   VAR
      s_FB_TRCV {InstructionName := 'TRCV'; LibVersion := '4.0'; ExternalAccessible := 'False'; ExternalVisible := 'False'; ExternalWritable := 'False'; S7_SetPoint := 'False'} : TRCV;   // Siemens "TRCV" block - to receive the data from TCPIP socket
      ss_TRCV { ExternalAccessible := 'False'; ExternalVisible := 'False'; ExternalWritable := 'False'} : Struct   // TRCV block interface structure
         Enable { ExternalAccessible := 'False'; ExternalVisible := 'False'; ExternalWritable := 'False'} : Bool;   //      TRCV - Enable
         NDR { ExternalAccessible := 'False'; ExternalVisible := 'False'; ExternalWritable := 'False'} : Bool;   //      TRCV - New data available
         Busy { ExternalAccessible := 'False'; ExternalVisible := 'False'; ExternalWritable := 'False'} : Bool;   //      TRCV - Busy
         Error { ExternalAccessible := 'False'; ExternalVisible := 'False'; ExternalWritable := 'False'} : Bool;   //      TRCV - Error
         Status { ExternalAccessible := 'False'; ExternalVisible := 'False'; ExternalWritable := 'False'} : Word;   //      TRCV - Status
         ReceivedLength { ExternalAccessible := 'False'; ExternalVisible := 'False'; ExternalWritable := 'False'} : UDInt;   //      TRCV - Received length
         Data { ExternalAccessible := 'False'; ExternalVisible := 'False'; ExternalWritable := 'False'} : Array[0..999] of Char;   //      TRCV - Data
      END_STRUCT;
      s_UDT_MessageArray { ExternalAccessible := 'False'; ExternalVisible := 'False'; ExternalWritable := 'False'; S7_SetPoint := 'False'} : "UDT_Message";   // Message byte array
      s_UDT_MessagePartArray { ExternalAccessible := 'False'; ExternalVisible := 'False'; ExternalWritable := 'False'; S7_SetPoint := 'False'} : "UDT_Message";   // Part of the message byte array
      ss_Status { ExternalAccessible := 'False'; ExternalVisible := 'False'; ExternalWritable := 'False'} : Struct   // Status structure
         ErrorCode { ExternalAccessible := 'False'; ExternalVisible := 'False'; ExternalWritable := 'False'} : Struct   // Error code structure
            TRCV { ExternalAccessible := 'False'; ExternalVisible := 'False'; ExternalWritable := 'False'} : Word;   //     Siemens TRCV error code - Check documentation
         END_STRUCT;
         FIFOReceiveStatus { ExternalAccessible := 'False'; ExternalVisible := 'False'; ExternalWritable := 'False'} : "UDT_FifoStatus";   // Receive FIFO status structure
         FIFOReceiveError { ExternalAccessible := 'False'; ExternalVisible := 'False'; ExternalWritable := 'False'; S7_SetPoint := 'True'} : Bool;   // Receive FIFO error
         FIFOReceiveWarning { ExternalAccessible := 'False'; ExternalVisible := 'False'; ExternalWritable := 'False'; S7_SetPoint := 'True'} : Bool;   // Receive  FIFO warning
         ReceiveError { ExternalAccessible := 'False'; ExternalVisible := 'False'; ExternalWritable := 'False'} : Bool;   // TRCV block operation error - Check TRCVStatus
      END_STRUCT;
      sui_ReceivedMessagesOffset { ExternalAccessible := 'False'; ExternalVisible := 'False'; ExternalWritable := 'False'} : Int;   // Received message offset
      sui_ReceivedMessageLength { ExternalAccessible := 'False'; ExternalVisible := 'False'; ExternalWritable := 'False'} : UInt;   // Received message length
      sui_NumberOfReceivedMessages { ExternalAccessible := 'False'; ExternalVisible := 'False'; ExternalWritable := 'False'} : UInt;   // Number of received messages in one frame
      sui_ReceivedMessagePartLength { ExternalAccessible := 'False'; ExternalVisible := 'False'; ExternalWritable := 'False'} : UInt;   // Length of the part of received message
      si_MaximumMessageLength { ExternalAccessible := 'False'; ExternalVisible := 'False'; ExternalWritable := 'False'} : Int;   // Maximum message length
      sx_ReceivedMessagePart { ExternalAccessible := 'False'; ExternalVisible := 'False'; ExternalWritable := 'False'} : Bool;   // Received part of the message
      sx_STXFound { ExternalAccessible := 'False'; ExternalVisible := 'False'; ExternalWritable := 'False'} : Bool;   // STX in message is found
   END_VAR

   VAR_TEMP
      ti_LC_MessageChars : Int;   //  Message chars loop counter
   END_VAR

   VAR CONSTANT
      cc_STX : Char := '$02';   // Start of the message sign
      cc_EXT : Char := '$03';   // End of the message sign
      cc_NULL : Char := '$00';   // Null sign
   END_VAR


BEGIN
	(*
	----------------------------------------------------------------------------------------

	Version history:
	Date        | Version   | Author        | Remark
	----------------------------------------------------------------------------------------
	25/10/2021  | 1.0       | J. Krawczuk   | Initial version TIA 16
	17/11/2021  | 1.2       | M. Piela      | Interface changes
	21/02/2023  | 4.0       | F.Baten       | 4.0 Release TIA 17.5
	13/03/2024  | 4.1       | S. Nieświec   | 4.1 Release TIA 18
	02/05/2024  | 4.2       | J.Majer      | Datatype conversions changed from automatic to explicit, to accomodate IEC 61131-3 standard
	*)

	REGION 1 – Update FIFO header status bits

	    // Mode 'S' - FIFO register status update.
	    "FC_Fifo"(ic_Mode := 'S',
	              qUDT_Status => #ss_Status.FIFOReceiveStatus,
	              qx_Error => #ss_Status.FIFOReceiveError,
	              qx_Warning => #ss_Status.FIFOReceiveWarning,
	              iqv_Data := #s_UDT_MessageArray,
	              iqUDT_FifoHeader := #iqUDT_FifoHeader,
	              iqv_DataBuffer := #iqv_FifoData);

	END_REGION

	REGION 2 – Maximum number of message arrays elements

	    #si_MaximumMessageLength := "FC_GetNrOfArrayEl"(iv_Array := #s_UDT_MessageArray.Character);

	END_REGION

	REGION 3 – Receive enable

	    // Allow receiving if the connection is established and there are no FIFO errors.
	    #ss_TRCV.Enable :=
	    #ix_EnableReceive
	    AND NOT #ss_Status.FIFOReceiveError;

	END_REGION

	REGION 4 – Receive data

	    // Data received in an ADHOC mode - data available immediately.
	    #s_FB_TRCV(EN_R := #ss_TRCV.Enable,
	               ID := #iUDT_Connection.ID,
	               LEN := 0,
	               ADHOC := TRUE,
	               NDR => #ss_TRCV.NDR,
	               BUSY => #ss_TRCV.Busy,
	               ERROR => #ss_TRCV.Error,
	               STATUS => #ss_TRCV.Status,
	               RCVD_LEN => #ss_TRCV.ReceivedLength,
	               DATA := #ss_TRCV.Data);

	END_REGION

	REGION 5 – Received data handling

	    // Receiving data was successful.
	    IF #ss_TRCV.NDR
	        AND NOT #ss_TRCV.Busy
	        AND NOT #ss_TRCV.Error
	        AND #ss_TRCV.ReceivedLength > 0

	    THEN

	        REGION 5.1 – Initialization

	            #sui_ReceivedMessageLength := 0;
	            #sui_ReceivedMessagesOffset := 0;
	            #sui_NumberOfReceivedMessages := 0;

	        END_REGION

	        REGION 5.2 – Received part of the message

	            // Move part of the messages into a buffer if available.
	            IF #sx_ReceivedMessagePart
	            THEN
	                #s_UDT_MessageArray := #s_UDT_MessagePartArray;
	            END_IF;

	        END_REGION

	        REGION 5.3 – Message handling

	            FOR #ti_LC_MessageChars := 0 TO (UDINT_TO_INT(#ss_TRCV.ReceivedLength) - 1) DO
	                // Message length validation.
	                IF #sui_ReceivedMessageLength <= #si_MaximumMessageLength
	                THEN
	                    // First termination sign found.
	                    IF (#ss_TRCV.Data[#ti_LC_MessageChars] = #cc_STX)
	                        AND NOT #sx_STXFound
	                    THEN
	                        #sx_STXFound := TRUE;
	                        #sui_ReceivedMessagesOffset := #ti_LC_MessageChars;

	                    ELSIF (#ss_TRCV.Data[#ti_LC_MessageChars] = #cc_STX)
	                        AND #sx_STXFound
	                    THEN
	                        // Increment invalid meassage statistic.
	                        #iqUDT_Statistics.InvalidMsg += 1;
	                        #sx_STXFound := FALSE;
	                    END_IF;

	                    // STX is found.
	                    IF #sx_STXFound
	                    THEN
	                        // Increment received message length.
	                        #sui_ReceivedMessageLength += 1;

	                        // End of the message sign is found.
	                        IF #ss_TRCV.Data[#ti_LC_MessageChars] = #cc_EXT
	                        THEN
	                            // Move received message to the message array.
	                            MOVE_BLK(IN := #ss_TRCV.Data[#sui_ReceivedMessagesOffset],
	                                     COUNT := #sui_ReceivedMessageLength,
	                                     OUT => #s_UDT_MessageArray.Character[#sui_ReceivedMessagePartLength]);

	                            // Clear not used message array characters.
	                            IF (#sui_ReceivedMessageLength + #sui_ReceivedMessagePartLength) < #si_MaximumMessageLength
	                            THEN
	                                FILL_BLK(IN := #cc_NULL,
	                                         COUNT := INT_TO_ULINT(#si_MaximumMessageLength) -
	                                         UDINT_TO_ULINT(#sui_ReceivedMessageLength) + #sui_ReceivedMessagePartLength,
	                                         OUT => #s_UDT_MessageArray.Character[#sui_ReceivedMessageLength + #sui_ReceivedMessagePartLength]);
	                            END_IF;

	                            // Mode 'W' - Write FIFO record.
	                            "FC_Fifo"(ic_Mode := 'W',
	                                      qUDT_Status => #ss_Status.FIFOReceiveStatus,
	                                      qx_Error => #ss_Status.FIFOReceiveError,
	                                      qx_Warning => #ss_Status.FIFOReceiveWarning,
	                                      iqv_Data := #s_UDT_MessageArray,
	                                      iqUDT_FifoHeader := #iqUDT_FifoHeader,
	                                      iqv_DataBuffer := #iqv_FifoData);

	                            // Increment received message count.
	                            #sui_NumberOfReceivedMessages += 1;
	                            // Initialize variables.
	                            #sui_ReceivedMessageLength := 0;
	                            #sui_ReceivedMessagePartLength := 0;
	                            #sx_ReceivedMessagePart := FALSE;
	                            #sx_STXFound := FALSE;

	                        END_IF;
	                    END_IF;
	                END_IF;
	            END_FOR;

	        END_REGION

	        REGION 5.4 – Part of the message preparation

	            // Only the part of the message is received.
	            IF (#ss_TRCV.Data[UDINT_TO_INT(#ss_TRCV.ReceivedLength) - 1] <> #cc_EXT            // Last received sign is not a termination sing
	                AND #sui_ReceivedMessageLength < #si_MaximumMessageLength)       // Message length valid
	                AND #sx_STXFound
	            THEN
	                // Clear not used message array characters.
	                FILL_BLK(IN := #cc_NULL,
	                         COUNT := INT_TO_ULINT(#si_MaximumMessageLength) -
	                         UDINT_TO_ULINT(#sui_ReceivedMessageLength),
	                         OUT => #s_UDT_MessagePartArray.Character[#sui_ReceivedMessageLength]);

	                // Move part of the message into a buffer.
	                MOVE_BLK(IN := #ss_TRCV.Data[#sui_ReceivedMessagesOffset],
	                         COUNT := #sui_ReceivedMessageLength,
	                         OUT => #s_UDT_MessagePartArray.Character[0]);

	                // Set the part of the message received bit and move length of the received message into the length of the part of the message variable.
	                #sx_ReceivedMessagePart := TRUE;
	                #sui_ReceivedMessagePartLength := #sui_ReceivedMessageLength;
	            END_IF;

	        END_REGION

	    END_IF;

	END_REGION

	REGION 6 – Status

	    REGION 6.1 - Block status

	        // Receive error.
	        #ss_Status.ReceiveError := #ss_TRCV.Error;

	        // Parametrization collective error output.
	        #qx_Error :=
	        #ss_Status.FIFOReceiveError
	        OR #ss_Status.ReceiveError;

	        // Parametrization collective warning output.
	        #qx_Warning := #ss_Status.FIFOReceiveWarning;

	    END_REGION

	    REGION 6.2 - Error code preparation

	        IF (#ss_TRCV.#Status > 16#8000)
	            OR (#ss_TRCV.#Status = 16#0)
	        THEN
	            #ss_Status.ErrorCode.TRCV := #ss_TRCV.#Status;
	        END_IF;

	    END_REGION
	END_REGION
END_FUNCTION_BLOCK

FUNCTION_BLOCK "FB_FedExHeartbeat"
TITLE = FB_Heartbeat
{ S7_Optimized_Access := 'TRUE' }
AUTHOR : MHSE
FAMILY : UPS_SpecificCommunication
VERSION : 3.0
// ATTRIBUTES
// AUTO_NUMBER = True
// BLOCK_NUMBER = 74
// END_ATTRIBUTES
//Function block to send and monitor the UPS heartbeat message.
   VAR_INPUT
      iudi_HeartbeatTimeout { ExternalAccessible := 'False'; ExternalVisible := 'False'; ExternalWritable := 'False'} : UDInt;   // Time after which block show heartbeat error
      iudi_HeartbeatInterval { ExternalAccessible := 'False'; ExternalVisible := 'False'; ExternalWritable := 'False'} : UDInt;   // Heartbeat send interval
      ix_Server { ExternalAccessible := 'False'; ExternalVisible := 'False'; ExternalWritable := 'False'} : Bool;   // PLC is Server ( True = Server )
      ix_EnableSend { ExternalAccessible := 'False'; ExternalVisible := 'False'; ExternalWritable := 'False'} : Bool;   // Enable heartbeat message send
      ix_ResetData { ExternalAccessible := 'False'; ExternalVisible := 'False'; ExternalWritable := 'False'} : Bool;   // Reset statistics
   END_VAR

   VAR_OUTPUT
      qx_HeartbeatOK { ExternalAccessible := 'False'; ExternalVisible := 'False'; ExternalWritable := 'False'} : Bool;   // Heartbeat ok
      qx_Error { ExternalAccessible := 'False'; ExternalVisible := 'False'; ExternalWritable := 'False'} : Bool;   // Collective error output
      qx_Warning { ExternalAccessible := 'False'; ExternalVisible := 'False'; ExternalWritable := 'False'} : Bool;   // Collective warning output
   END_VAR

   VAR_IN_OUT
      iqUDT_FifoHeader : "UDT_FifoHeader";   // FIFO header
      iqa_FifoData : Array[*] of "UDT_Message";   // FIFO data
      iqUDT_Statistics : "UDT_FedExHeartbeatStatistics";   // Heartbeat Statistics
      iqx_Heartbeat { ExternalAccessible := 'False'; ExternalVisible := 'False'; ExternalWritable := 'False'} : Bool;   // Heartbreat received
      iqx_ResetWritingTimer { ExternalAccessible := 'False'; ExternalVisible := 'False'; ExternalWritable := 'False'} : Bool;   // Any message received, do not send Heartbeat
      iqx_ResetListeningTimer { ExternalAccessible := 'False'; ExternalVisible := 'False'; ExternalWritable := 'False'} : Bool;   // Any message received, reset timeout timer
      iqx_SendLS { ExternalAccessible := 'False'; ExternalVisible := 'False'; ExternalWritable := 'False'} : Bool;   // Close the connection
      iqx_Reconnect { ExternalAccessible := 'False'; ExternalVisible := 'False'; ExternalWritable := 'False'} : Bool;   // Reconnect command
   END_VAR

   VAR
      sR_TRIG_EnableSend {InstructionName := 'R_TRIG'; LibVersion := '1.0'; ExternalAccessible := 'False'; ExternalVisible := 'False'; ExternalWritable := 'False'; S7_SetPoint := 'False'} : R_TRIG;   // Siemens "R_TRIG" - to prepare the rising edge trigger on "ix_EnableSend" signal
      sUDT_MessageArray { ExternalAccessible := 'False'; ExternalVisible := 'False'; ExternalWritable := 'False'; S7_SetPoint := 'False'} : "UDT_Message";   // Message character array
      sa_Status { ExternalAccessible := 'False'; ExternalVisible := 'False'; ExternalWritable := 'False'} : Struct   // Status structure
         FIFOStatus { ExternalAccessible := 'False'; ExternalVisible := 'False'; ExternalWritable := 'False'} : "UDT_FifoStatus";
         FIFOError { ExternalAccessible := 'False'; ExternalVisible := 'False'; ExternalWritable := 'False'; S7_SetPoint := 'True'} : Bool;   // FIFO data buffer full
         FIFOWarning { ExternalAccessible := 'False'; ExternalVisible := 'False'; ExternalWritable := 'False'; S7_SetPoint := 'True'} : Bool;   // FIFO error
         HeartbeatOk { ExternalAccessible := 'False'; ExternalVisible := 'False'; ExternalWritable := 'False'} : Bool;   // FIFO warning
         InvalidTimeInterval { ExternalAccessible := 'False'; ExternalVisible := 'False'; ExternalWritable := 'False'} : Bool;   // Heartbeat ok
         InvalidTimeout { ExternalAccessible := 'False'; ExternalVisible := 'False'; ExternalWritable := 'False'} : Bool;   // Heartbeat time interval lower than zero
         InvalidMsgArraySize { ExternalAccessible := 'False'; ExternalVisible := 'False'; ExternalWritable := 'False'} : Bool;   // Heartbeat timeout lower than zero or lower than heartbeat time interval
      END_STRUCT;
      sFB_HeartbeatPulse { ExternalAccessible := 'False'; ExternalVisible := 'False'; ExternalWritable := 'False'; S7_SetPoint := 'False'} : "FB_TimerOnOffDelay";   // Sending Heartbeat timer
      sFB_Timer_HeartbeatCheck { ExternalAccessible := 'False'; ExternalVisible := 'False'; ExternalWritable := 'False'; S7_SetPoint := 'False'} : "FB_TimerOnOffDelay";   // MHS "FB_TimerOnOffDelay" - to measure the time of  missing Hearbeat
      ss_Message { ExternalAccessible := 'False'; ExternalVisible := 'False'; ExternalWritable := 'False'} : String;   // Message character string
      sui_MsgArrayElNr { ExternalAccessible := 'False'; ExternalVisible := 'False'; ExternalWritable := 'False'} : UInt;   // Invalid message array size
      si_MaxMsgLen { ExternalAccessible := 'False'; ExternalVisible := 'False'; ExternalWritable := 'False'} : Int;   // Maximum message length
      si_MsgLen { ExternalAccessible := 'False'; ExternalVisible := 'False'; ExternalWritable := 'False'} : Int;   // String character message length
      si_LostMsg { ExternalAccessible := 'False'; ExternalVisible := 'False'; ExternalWritable := 'False'} : Int;   // Number of lost heartbeat messages
      sx_HeartbeatPulse { ExternalAccessible := 'False'; ExternalVisible := 'False'; ExternalWritable := 'False'} : Bool;   // Heartbeat pulse
      sx_HeartbeatOk { ExternalAccessible := 'False'; ExternalVisible := 'False'; ExternalWritable := 'False'} : Bool;   // Heartbeat ok
      sx_MsgLost { ExternalAccessible := 'False'; ExternalVisible := 'False'; ExternalWritable := 'False'} : Bool;   // Message lost
      sx_HeartbeatCheck { ExternalAccessible := 'False'; ExternalVisible := 'False'; ExternalWritable := 'False'} : Bool;   // Heartbeat check
   END_VAR

   VAR CONSTANT
      cc_STX : Char := '$02';   // Start of the text
      cc_ETX : Char := '$03';   // End of the text
      cc_NULL : Char := '$00';   // NULL sign
      cs_Length : String := '0006';   // Legth of the message
      cs_MessageType : String := 'HB';   // Message type
   END_VAR


BEGIN
	(*
	----------------------------------------------------------------------------------------

	Version history:
	Date        | Version   | Author        | Remark
	----------------------------------------------------------------------------------------
	29/06/2021  | 0.1       | F.Baten       | First release 16.0
	05/04/2022  | 0.2       | K.Pokorski    | Review
	21/02/2023  | 4.0       | F.Baten       | 4.0 Release TIA 17.5
	*)

	REGION 1 – FIFO header status update

	    // Mode 'S' - FIFO register status update
	    "FC_Fifo"(ic_Mode := 'S',
	              qUDT_Status => #sa_Status.FIFOStatus,
	              qx_Error => #sa_Status.FIFOError,
	              qx_Warning => #sa_Status.FIFOWarning,
	              iqv_Data := #sUDT_MessageArray,
	              iqUDT_FifoHeader := #iqUDT_FifoHeader,
	              iqv_DataBuffer := #iqa_FifoData);


	END_REGION

	REGION 2 – Heartbeat time interval and timeout validation
	    IF NOT #ix_Server
	    THEN
	        #sa_Status.InvalidTimeInterval := #iudi_HeartbeatInterval <= 0;

	        #sa_Status.InvalidTimeout := #iudi_HeartbeatTimeout <= 0
	        OR #iudi_HeartbeatTimeout <= #iudi_HeartbeatInterval;
	    END_IF;

	END_REGION

	REGION 3 – Heartbeat pulse generation

	    IF (NOT #sa_Status.InvalidTimeInterval                  // Preset heartbeat time interval is valid
	        AND NOT #sa_Status.InvalidTimeout)                  // Timeout is valid
	        AND NOT #ix_Server
	    THEN

	        #sFB_HeartbeatPulse(iudi_OnDelayTime := #iudi_HeartbeatInterval,
	                            iudi_OffDelayTime := 0,
	                            ix_SignalToDelay := NOT #iqx_ResetWritingTimer,
	                            qx_DelayedSignal => #sx_HeartbeatPulse);

	        IF #sx_HeartbeatPulse THEN
	            #iqx_ResetWritingTimer := TRUE;
	        ELSE
	            #iqx_ResetWritingTimer := FALSE;
	        END_IF;

	    END_IF;

	    // Reset heartbeat send request if PLC is a server
	    IF #ix_Server
	    THEN
	        #sx_HeartbeatPulse := #iqx_Heartbeat;
	        //  #iqx_Heartbeat := FALSE;
	    END_IF;
	END_REGION

	REGION 4 – Heartbeat message preparation

	    IF (NOT #iqUDT_FifoHeader.Status.Full)                 // FIFO isn't full
	    THEN

	        IF (#sx_HeartbeatPulse                              // Heartbeat pulse available
	            AND #ix_EnableSend                              // Send is enable
	            AND NOT #sa_Status.FIFOError)                   // No FIFO error
	        THEN
	            REGION 4.1 – Message preparation

	                // Heartbeat message composing according to the structure: STX,00,06,HB,ETX
	                #ss_Message := CONCAT(IN1 := #cc_STX,               // Start of message
	                                      IN2 := #cs_Length,            // message length
	                                      IN3 := #cs_MessageType,       // Heartbeat
	                                      IN4 := #cc_ETX);              // End of message

	            END_REGION

	            REGION 4.2 – Maximum number of the message characters

	                #si_MaxMsgLen := "FC_GetNrOfArrayEl"(iv_Array := #sUDT_MessageArray.Character);

	            END_REGION

	            REGION 4.3 – Length of the complete message

	                #si_MsgLen := LEN(#ss_Message);

	            END_REGION

	            REGION 4.4 –  Message array size validation

	                #sa_Status.InvalidMsgArraySize := #si_MsgLen > #si_MaxMsgLen;

	            END_REGION

	            REGION 4.5 –  Message character string conversion to a message array of characters

	                IF (NOT #sa_Status.InvalidMsgArraySize)     // Message character array size is valid
	                THEN

	                    Strg_TO_Chars(Strg := #ss_Message,
	                                  pChars := 0,
	                                  Cnt => #sui_MsgArrayElNr,
	                                  Chars := #sUDT_MessageArray.Character);

	                END_IF;

	            END_REGION

	            REGION 4.6 – Clearing remaining characters in the message character array

	                IF (NOT #sa_Status.InvalidMsgArraySize)     // Message character array size is valid
	                THEN

	                    // Filling up not used message character array elements with '$00' (ASCII - 16#00)
	                    FILL_BLK(IN := #cc_NULL,
	                             COUNT := UINT_TO_ULINT(INT_TO_UINT(#si_MaxMsgLen) - #sui_MsgArrayElNr),
	                             OUT => #sUDT_MessageArray.Character[#sui_MsgArrayElNr]);

	                END_IF;

	            END_REGION

	            REGION 4.7 – Message write into a FIFO register

	                IF (#ix_EnableSend                          // Heartbeat send enable
	                    AND NOT #sa_Status.InvalidMsgArraySize) // Message character array size is valid
	                THEN

	                    // Mode 'W' - Write FIFO record
	                    "FC_Fifo"(ic_Mode := 'W',
	                              qUDT_Status => #sa_Status.FIFOStatus,
	                              qx_Error => #sa_Status.FIFOError,
	                              qx_Warning => #sa_Status.FIFOWarning,
	                              iqv_Data := #sUDT_MessageArray,
	                              iqUDT_FifoHeader := #iqUDT_FifoHeader,
	                              iqv_DataBuffer := #iqa_FifoData);
	                END_IF;

	            END_REGION

	        END_IF;

	        // In case of FIFO full, the FIFO full error bit and FIFO collective error bit are set
	    ELSE

	        #sa_Status.FIFOError := TRUE;
	        #sa_Status.FIFOStatus.FifoFull := TRUE;

	    END_IF;

	END_REGION

	REGION 5 – Heartbeat monitoring
	    // IF NOT #ix_Server
	    // THEN
	    IF (NOT #sa_Status.InvalidTimeInterval                  // Time interval is valid
	        AND NOT #sa_Status.InvalidTimeout                   // Timeout is  valid
	        AND NOT #sa_Status.InvalidMsgArraySize)             // Message character array size is valid

	    THEN

	        #sR_TRIG_EnableSend(CLK := #ix_EnableSend);

	        // Reset heartbeat ok
	        IF (NOT #ix_EnableSend)                             // Heartbeat send not enable
	        THEN
	            #iqx_SendLS := FALSE;
	            #sx_HeartbeatOk := FALSE;

	        END_IF;

	        // Clear auxiliary variables
	        IF (#iqx_Heartbeat                                  // Hearbeat message received
	            AND #ix_EnableSend)                             // Heartbeat send enable
	        THEN

	            #si_LostMsg := 0;                               // Lost messages counter
	            #sx_MsgLost := FALSE;                           // Message lost bit
	            #sx_HeartbeatOk := TRUE;                        // HeartbeatOk bit

	        END_IF;

	        // Time measurement of a missing heartbeat
	        #sFB_Timer_HeartbeatCheck(ix_SignalToDelay := #iqx_Heartbeat           // Heartbeat signal
	                                  OR #sx_MsgLost                               // Message lost
	                                  OR #sR_TRIG_EnableSend.Q                    // Enable send trigger
	                                  OR #iqx_ResetListeningTimer,                 // Any message received in this socket
	                                  iudi_OnDelayTime := 0,
	                                  iudi_OffDelayTime := #iudi_HeartbeatTimeout,
	                                  qx_DelayedSignal => #sx_HeartbeatCheck);

	        #iqx_Heartbeat := FALSE;
	        #sx_MsgLost := FALSE;
	        #iqx_ResetListeningTimer := FALSE;

	        // Increment lost messages counter and set lost message bit
	        IF (NOT #sx_HeartbeatCheck                          // Heartbeat not checked
	            AND NOT #iqx_Reconnect                          // No reconnect command
	            AND #ix_EnableSend)                             // Send is enable
	        THEN

	            // Send LS, re-establish connection, increment statistics and signalize heartbeat error

	            #iqx_SendLS := TRUE;
	            #iqUDT_Statistics.ConLost += 1;
	            #si_LostMsg := 0;
	            #sx_MsgLost := FALSE;
	            #sx_HeartbeatOk := FALSE;

	        END_IF;

	        // Configuration error occured
	    ELSE

	        #sx_HeartbeatOk := FALSE;

	    END_IF;
	    // END_IF;

	END_REGION

	REGION 6 – Statistics

	    IF #iqUDT_FifoHeader.Status.Full
	        AND #sx_HeartbeatPulse
	    THEN
	        #iqUDT_Statistics.MsgNotSent += 1;

	    END_IF;

	    IF (#ix_ResetData)                                      // Reset statistics request
	    THEN
	        #iqUDT_Statistics.ConLost := 0;
	        #iqUDT_Statistics.MsgNotSent := 0;

	    END_IF;

	END_REGION

	REGION 7 – Status

	    // Hearbeat ok output
	    #qx_HeartbeatOK := #sx_HeartbeatOk;

	    // Parametrization collective error output
	    #qx_Error :=
	    #sa_Status.InvalidTimeInterval                          // Invalid time interval
	    OR #sa_Status.InvalidTimeout                            // Invalid timeout
	    OR #sa_Status.InvalidMsgArraySize                       // Invalid message character array size
	    OR #sa_Status.FIFOError                                 // FIFO error
	    OR NOT #sx_HeartbeatOk;                                 // No heartbeat OK

	    // Parametrization collective warning output
	    #qx_Warning := #sa_Status.FIFOWarning;                  // FIFO warning

	END_REGION
END_FUNCTION_BLOCK

FUNCTION_BLOCK "FB_FedExDecode"
TITLE = FB_Decode
{ S7_Optimized_Access := 'TRUE' }
AUTHOR : MHSE
FAMILY : UPS_SpecificCommunication
VERSION : 3.0
// ATTRIBUTES
// AUTO_NUMBER = True
// BLOCK_NUMBER = 65
// END_ATTRIBUTES
//Function block to decode UPS messages.
   VAR_IN_OUT
      iqUDT_FifoRcvHeader : "UDT_FifoHeader";   // FIFO receive header
      iqv_FifoRcvData : Array[*] of "UDT_Message";   // FIFO receive data
      iqx_HeartbeatOk { ExternalAccessible := 'False'; ExternalVisible := 'False'; ExternalWritable := 'False'} : Bool;   // Heartbeat signal was received
   END_VAR

   VAR
      sUDT_MSGHeader { ExternalAccessible := 'False'; ExternalVisible := 'False'; ExternalWritable := 'False'; S7_SetPoint := 'False'} : "UDT_FedExMessageHeader";
      sUDT_SI { ExternalAccessible := 'False'; ExternalVisible := 'False'; ExternalWritable := 'False'; S7_SetPoint := 'False'} : "UDT_FedExMessageSI";
      sUDT_WS { ExternalAccessible := 'False'; ExternalVisible := 'False'; ExternalWritable := 'False'; S7_SetPoint := 'False'} : "UDT_FedExMessageWS";
      sUDT_DA { ExternalAccessible := 'False'; ExternalVisible := 'False'; ExternalWritable := 'False'; S7_SetPoint := 'False'} : "UDT_FedExMessageDaRa";
      sUDT_RA { ExternalAccessible := 'False'; ExternalVisible := 'False'; ExternalWritable := 'False'; S7_SetPoint := 'False'} : "UDT_FedExMessageDaRa";
      sUDT_FifoMsg { ExternalAccessible := 'False'; ExternalVisible := 'False'; ExternalWritable := 'False'; S7_SetPoint := 'False'} : "UDT_Message";   // Buffer for fifos message
      sa_Status { ExternalAccessible := 'False'; ExternalVisible := 'False'; ExternalWritable := 'False'} : Struct   // Status structure
         BadMessage { ExternalAccessible := 'False'; ExternalVisible := 'False'; ExternalWritable := 'False'} : Array[1..10] of "UDT_Message";   //   Unknown message read
         FIFORcvStatus { ExternalAccessible := 'False'; ExternalVisible := 'False'; ExternalWritable := 'False'} : "UDT_FifoStatus";   //   Receive FIFO status structure
         FIFOError { ExternalAccessible := 'False'; ExternalVisible := 'False'; ExternalWritable := 'False'; S7_SetPoint := 'True'} : Bool;   //   FIFO error
         FIFOWarning { ExternalAccessible := 'False'; ExternalVisible := 'False'; ExternalWritable := 'False'; S7_SetPoint := 'True'} : Bool;   //   FIFO warning
         AcknowledgeError { ExternalAccessible := 'False'; ExternalVisible := 'False'; ExternalWritable := 'False'; S7_SetPoint := 'True'} : Bool;   //   Acknowledge error
         AcknowledgeWarning { ExternalAccessible := 'False'; ExternalVisible := 'False'; ExternalWritable := 'False'; S7_SetPoint := 'True'} : Bool;   //   Acknowledge warning
         HB_NotOK { ExternalAccessible := 'False'; ExternalVisible := 'False'; ExternalWritable := 'False'} : Bool;   //   Health bit not OK
      END_STRUCT;
      ss_NNNNNN { ExternalAccessible := 'False'; ExternalVisible := 'False'; ExternalWritable := 'False'} : String[6];
      sdi_DeserializePosition { ExternalAccessible := 'False'; ExternalVisible := 'False'; ExternalWritable := 'False'} : DInt;
      si_DeserializeBodyStatus { ExternalAccessible := 'False'; ExternalVisible := 'False'; ExternalWritable := 'False'} : Int;
      si_Length { ExternalAccessible := 'False'; ExternalVisible := 'False'; ExternalWritable := 'False'} : Int;
      si_Position { ExternalAccessible := 'False'; ExternalVisible := 'False'; ExternalWritable := 'False'} : Int;   // Temporary position parial message
      si_SizeOfMsg { ExternalAccessible := 'False'; ExternalVisible := 'False'; ExternalWritable := 'False'} : Int;   // Message array size
      si_GIN { ExternalAccessible := 'False'; ExternalVisible := 'False'; ExternalWritable := 'False'} : Int;
      sx_InvalidLength { ExternalAccessible := 'False'; ExternalVisible := 'False'; ExternalWritable := 'False'} : Bool;
   END_VAR

   VAR_TEMP
      tx_MsgRead : Bool;   // Message read from FIFO
   END_VAR

   VAR CONSTANT
      cs_SI : String := 'SI';
      cs_WS : String := 'WS';
      cs_DA : String := 'DA';
      cs_RA : String := 'RA';
      cs_ES : String := 'ES';
      cs_HB : String := 'HB';
      ci_SizeSIMessage : Int := 338;
      ci_SizeWSMessage : Int := 92;
      ci_SizeDAMessage : Int := 212;
      ci_SizeRAMessage : Int := 212;
      ci_SizeESMessage : Int := 57;
   END_VAR


BEGIN
	(*
	----------------------------------------------------------------------------------------

	Version history:
	Date        | Version   | Author        | Remark
	----------------------------------------------------------------------------------------
	22/07/2021  | 0.1       | F.Baten       | first release MHS TIA 15.1
	21/02/2023  | 4.0       | F.Baten       | 4.0 Release TIA 17.5
	*)

	REGION 1 – FIFO header status update

	    // Mode 'S' - FIFO register status update
	    "FC_Fifo"(ic_Mode := 'S',
	              qUDT_Status => #sa_Status.FIFORcvStatus,
	              qx_Error => #sa_Status.FIFOError,
	              qx_Warning => #sa_Status.FIFOWarning,
	              iqv_Data := #sUDT_FifoMsg,
	              iqUDT_FifoHeader := #iqUDT_FifoRcvHeader,
	              iqv_DataBuffer := #iqv_FifoRcvData);

	    IF (NOT #iqUDT_FifoRcvHeader.Status.Empty                             // FIFO not empty
	        AND NOT #sa_Status.FIFOError)                                      // No FIFO error
	    THEN

	        // Mode 'R' - Read FIFO record
	        "FC_Fifo"(ic_Mode := 'R',
	                  qUDT_Status => #sa_Status.FIFORcvStatus,
	                  qx_Error => #sa_Status.FIFOError,
	                  qx_Warning => #sa_Status.FIFOWarning,
	                  iqv_Data := #sUDT_FifoMsg,
	                  iqUDT_FifoHeader := #iqUDT_FifoRcvHeader,
	                  iqv_DataBuffer := #iqv_FifoRcvData);

	        // Message read bit set and position initialize
	        #tx_MsgRead := TRUE;
	        #si_Position := 0;

	        // FIFO empty or FIFO error occured
	    ELSE

	        #tx_MsgRead := FALSE;

	    END_IF;

	END_REGION

	REGION 1 – Maximum number of the message characters

	    #si_SizeOfMsg := "FC_GetNrOfArrayEl"(iv_Array := #sUDT_FifoMsg.Character);


	END_REGION

	REGION 2 – Decoding header
	    #sUDT_MSGHeader.MessageType := '';

	    IF #tx_MsgRead
	    THEN
	        // Converting message header from array of bytes to UDT.

	        #sdi_DeserializePosition := 0;
	        #si_DeserializeBodyStatus := Deserialize(SRC_ARRAY := #sUDT_FifoMsg,
	                                                 DEST_VARIABLE => #sUDT_MSGHeader,
	                                                 POS := #sdi_DeserializePosition);
	        // Character length into integer conversion
	        #si_Length := STRING_TO_INT(IN := #sUDT_MSGHeader.MessageLength);
	    END_IF;
	END_REGION

	REGION 3 - decode Scan Information
	    // Message is read and type is SI
	    IF #tx_MsgRead
	        AND #sUDT_MSGHeader.MessageType = #cs_SI
	    THEN
	        // Convert array of bytes into body structure.
	        #si_DeserializeBodyStatus := Deserialize(SRC_ARRAY := #sUDT_FifoMsg,
	                                                 DEST_VARIABLE => #sUDT_SI,
	                                                 POS := #sdi_DeserializePosition);
	        // Message length is fixed and should be the same
	        IF #si_Length <> #ci_SizeSIMessage
	        THEN
	            #sx_InvalidLength := TRUE;
	        ELSE
	            #sx_InvalidLength := FALSE;
	        END_IF;
	        IF NOT #sx_InvalidLength
	        THEN
	            // Convert 'NNNNNN' part in package ID to GIN number and store data in GIN database
	            #ss_NNNNNN := RIGHT(IN := #sUDT_SI.PackageID, L := 6);
	            STRG_VAL(IN := #ss_NNNNNN,
	                     FORMAT := 16#0,
	                     P := 1,
	                     OUT => #si_GIN);

	            "DB_GIN".GIN[#si_GIN].FedEx.ADCSystemID := #sUDT_SI.ADCSystemID;
	            "DB_GIN".GIN[#si_GIN].FedEx.ScanUnitType := #sUDT_SI.ScanUnitType;
	            "DB_GIN".GIN[#si_GIN].FedEx.ImageID := #sUDT_SI.ImageID;
	            "DB_GIN".GIN[#si_GIN].FedEx.PackageID := #sUDT_SI.PackageID;
	            "DB_GIN".GIN[#si_GIN].FedEx.HLCPackageID := #sUDT_SI.HLCPackageID;
	            "DB_GIN".GIN[#si_GIN].FedEx.DIMSystemID := #sUDT_SI.DIMSystemID;
	            "DB_GIN".GIN[#si_GIN].FedEx.DIMStatus := #sUDT_SI.DimStatus;
	            "DB_GIN".GIN[#si_GIN].FedEx.PackageDimLength := #sUDT_SI.PackageDimLength;
	            "DB_GIN".GIN[#si_GIN].FedEx.PackageDimWidth := #sUDT_SI.PackageDimWidth;
	            "DB_GIN".GIN[#si_GIN].FedEx.PackageDimHeight := #sUDT_SI.PackageDimHeight;
	            "DB_GIN".GIN[#si_GIN].FedEx.DIMUOM := #sUDT_SI.DIMUOM;
	            "DB_GIN".GIN[#si_GIN].FedEx.DimLFTstatusCode := #sUDT_SI.DimLFTstatusCode;
	            "DB_GIN".GIN[#si_GIN].FedEx.AlibiDims := #sUDT_SI.AlibiDims;
	            "DB_GIN".GIN[#si_GIN].FedEx.SCLSystemID := #sUDT_SI.SCLSystemID;
	            "DB_GIN".GIN[#si_GIN].FedEx.SCLStatus := #sUDT_SI.SCLStatus;
	            "DB_GIN".GIN[#si_GIN].FedEx.SCLWT := #sUDT_SI.SCLWT;
	            "DB_GIN".GIN[#si_GIN].FedEx.SCLWTUOM := #sUDT_SI.SCLWTUOM;
	            "DB_GIN".GIN[#si_GIN].FedEx.SCLLFTStatusCode := #sUDT_SI.SCLLFTStatusCode;
	            "DB_GIN".GIN[#si_GIN].FedEx.AlibiWeight := #sUDT_SI.AlibiWeight;
	            "DB_GIN".GIN[#si_GIN].FedEx.Stackable := #sUDT_SI.Stackable;
	            "DB_GIN".GIN[#si_GIN].FedEx.CameraHeadstatus := #sUDT_SI.CameraHeadstatus;
	            "DB_GIN".GIN[#si_GIN].FedEx.PackageDataTruncated := #sUDT_SI.PackageDataTruncated;
	            "DB_GIN".GIN[#si_GIN].FedEx.TotalBarcodeDataLength := #sUDT_SI.TotalBarcodeDataLength;
	            "DB_GIN".GIN[#si_GIN].FedEx.Barcode1Identification := #sUDT_SI.Barcode1Identification;
	            "DB_GIN".GIN[#si_GIN].FedEx.Barcode1status := #sUDT_SI.Barcode1status;
	            "DB_GIN".GIN[#si_GIN].FedEx.Barcode1datalength := #sUDT_SI.Barcode1datalength;
	            "DB_GIN".GIN[#si_GIN].FedEx.Barcode1data := #sUDT_SI.Barcode1data;
	            "DB_GIN".GIN[#si_GIN].FedEx.Barcode2Identification := #sUDT_SI.Barcode2Identification;
	            "DB_GIN".GIN[#si_GIN].FedEx.Barcode2status := #sUDT_SI.Barcode2status;
	            "DB_GIN".GIN[#si_GIN].FedEx.Barcode2datalength := #sUDT_SI.Barcode2datalength;
	            "DB_GIN".GIN[#si_GIN].FedEx.Barcode2data := #sUDT_SI.Barcode2data;
	            "DB_GIN".GIN[#si_GIN].FedEx.Barcode3Identification := #sUDT_SI.Barcode3Identification;
	            "DB_GIN".GIN[#si_GIN].FedEx.Barcode3status := #sUDT_SI.Barcode3status;
	            "DB_GIN".GIN[#si_GIN].FedEx.Barcode3datalength := #sUDT_SI.Barcode3datalength;
	            "DB_GIN".GIN[#si_GIN].FedEx.Barcode3data := #sUDT_SI.Barcode3data;
	        END_IF;
	    END_IF;
	END_REGION

	REGION 4 - Decode Weight Scale Message
	    // Message is read and type is WS
	    IF #tx_MsgRead
	        AND #sUDT_MSGHeader.MessageType = #cs_WS
	    THEN
	        // Convert array of bytes into body structure.
	        #si_DeserializeBodyStatus := Deserialize(SRC_ARRAY := #sUDT_FifoMsg,
	                                                 DEST_VARIABLE => #sUDT_WS,
	                                                 POS := #sdi_DeserializePosition);
	        // Message length is fixed and should be the same
	        IF #si_Length <> #ci_SizeWSMessage
	        THEN
	            #sx_InvalidLength := TRUE;
	        ELSE
	            #sx_InvalidLength := FALSE;
	        END_IF;
	        IF NOT #sx_InvalidLength
	        THEN
	            // Convert 'NNNNNN' part in package ID to GIN number and store data in GIN database
	            #ss_NNNNNN := RIGHT(IN := #sUDT_WS.PackageID, L := 6);
	            STRG_VAL(IN := #ss_NNNNNN,
	                     FORMAT := 16#0,
	                     P := 1,
	                     OUT => #si_GIN);

	            "DB_GIN".GIN[#si_GIN].FedEx.SCLSystemID := #sUDT_WS.SCLSystemID;
	            "DB_GIN".GIN[#si_GIN].FedEx.SCLWT := #sUDT_WS.SCLWT;
	            "DB_GIN".GIN[#si_GIN].FedEx.SCLWTUOM := #sUDT_WS.SCLWTUOM;
	            "DB_GIN".GIN[#si_GIN].FedEx.SCLLFTStatusCode := #sUDT_WS.SCLLFTStatusCode;
	            "DB_GIN".GIN[#si_GIN].FedEx.AlibiWeight := #sUDT_WS.AlibiWeight;
	        END_IF;
	    END_IF;
	END_REGION

	REGION 5 - Decode Destination Assignment message
	    // Message is read and type is DA
	    IF #tx_MsgRead
	        AND #sUDT_MSGHeader.MessageType = #cs_DA
	    THEN
	        // Convert array of bytes into body structure.
	        #si_DeserializeBodyStatus := Deserialize(SRC_ARRAY := #sUDT_FifoMsg,
	                                                 DEST_VARIABLE => #sUDT_DA,
	                                                 POS := #sdi_DeserializePosition);
	        // Message length is fixed and should be the same
	        IF #si_Length <> #ci_SizeDAMessage
	            OR #si_Length <> #si_SizeOfMsg
	        THEN
	            #sx_InvalidLength := TRUE;
	        ELSE
	            #sx_InvalidLength := FALSE;
	        END_IF;
	        IF NOT #sx_InvalidLength
	        THEN
	            // Convert 'NNNNNN' part in package ID to GIN number and store data in GIN database
	            #ss_NNNNNN := RIGHT(IN := #sUDT_DA.PackageID, L := 6);
	            STRG_VAL(IN := #ss_NNNNNN,
	                     FORMAT := 16#0,
	                     P := 1,
	                     OUT => #si_GIN);

	            "DB_GIN".GIN[#si_GIN].FedEx.HLCPackageID := #sUDT_DA.HLCPackageID;
	            "DB_GIN".GIN[#si_GIN].FedEx.CellNumber := #sUDT_DA.CellNumber;
	            "DB_GIN".GIN[#si_GIN].FedEx.Destination1 := #sUDT_DA.Destination1;
	            "DB_GIN".GIN[#si_GIN].FedEx.CutOffTimeDestination1 := #sUDT_DA.CutOffTimeDestination1;
	            "DB_GIN".GIN[#si_GIN].FedEx.Destination2 := #sUDT_DA.Destination2;
	            "DB_GIN".GIN[#si_GIN].FedEx.CutOffTimeDestination2 := #sUDT_DA.CutOffTimeDestination2;
	            "DB_GIN".GIN[#si_GIN].FedEx.Destination3 := #sUDT_DA.Destination3;
	            "DB_GIN".GIN[#si_GIN].FedEx.CutOffTimeDestination3 := #sUDT_DA.CutOffTimeDestination3;
	            "DB_GIN".GIN[#si_GIN].FedEx.Destination4 := #sUDT_DA.Destination4;
	            "DB_GIN".GIN[#si_GIN].FedEx.CutOffTimeDestination4 := #sUDT_DA.CutOffTimeDestination4;
	            "DB_GIN".GIN[#si_GIN].FedEx.Destination5 := #sUDT_DA.Destination5;
	            "DB_GIN".GIN[#si_GIN].FedEx.CutOffTimeDestination5 := #sUDT_DA.CutOffTimeDestination5;
	            "DB_GIN".GIN[#si_GIN].FedEx.HLCDataText := #sUDT_DA.HLCDataText;
	            "DB_GIN".GIN[#si_GIN].FedEx.Barcodedata := #sUDT_DA.Barcodedata;
	            "DB_GIN".GIN[#si_GIN].FedEx.HLCResultCode := #sUDT_DA.HLCResultCode;
	        END_IF;
	    END_IF;
	END_REGION

	REGION 6 - Decode destination Re-Assignment message
	    // Message is read and type is RA
	    IF #tx_MsgRead
	        AND #sUDT_MSGHeader.MessageType = #cs_RA
	    THEN
	        // Convert array of bytes into body structure.
	        #si_DeserializeBodyStatus := Deserialize(SRC_ARRAY := #sUDT_FifoMsg,
	                                                 DEST_VARIABLE => #sUDT_RA,
	                                                 POS := #sdi_DeserializePosition);
	        // Message length is fixed and should be the same
	        IF #si_Length <> #ci_SizeRAMessage
	            OR #si_Length <> #si_SizeOfMsg
	        THEN
	            #sx_InvalidLength := TRUE;
	        ELSE
	            #sx_InvalidLength := FALSE;
	        END_IF;
	        IF NOT #sx_InvalidLength
	        THEN
	            // Convert 'NNNNNN' part in package ID to GIN number and store data in GIN database
	            #ss_NNNNNN := RIGHT(IN := #sUDT_RA.PackageID, L := 6);
	            STRG_VAL(IN := #ss_NNNNNN,
	                     FORMAT := 16#0,
	                     P := 1,
	                     OUT => #si_GIN);

	            "DB_GIN".GIN[#si_GIN].FedEx.HLCPackageID := #sUDT_RA.HLCPackageID;
	            "DB_GIN".GIN[#si_GIN].FedEx.CellNumber := #sUDT_RA.CellNumber;
	            "DB_GIN".GIN[#si_GIN].FedEx.Destination1 := #sUDT_RA.Destination1;
	            "DB_GIN".GIN[#si_GIN].FedEx.CutOffTimeDestination1 := #sUDT_RA.CutOffTimeDestination1;
	            "DB_GIN".GIN[#si_GIN].FedEx.Destination2 := #sUDT_RA.Destination2;
	            "DB_GIN".GIN[#si_GIN].FedEx.CutOffTimeDestination2 := #sUDT_RA.CutOffTimeDestination2;
	            "DB_GIN".GIN[#si_GIN].FedEx.Destination3 := #sUDT_RA.Destination3;
	            "DB_GIN".GIN[#si_GIN].FedEx.CutOffTimeDestination3 := #sUDT_RA.CutOffTimeDestination3;
	            "DB_GIN".GIN[#si_GIN].FedEx.Destination4 := #sUDT_RA.Destination4;
	            "DB_GIN".GIN[#si_GIN].FedEx.CutOffTimeDestination4 := #sUDT_RA.CutOffTimeDestination4;
	            "DB_GIN".GIN[#si_GIN].FedEx.Destination5 := #sUDT_RA.Destination5;
	            "DB_GIN".GIN[#si_GIN].FedEx.CutOffTimeDestination5 := #sUDT_RA.CutOffTimeDestination5;
	            "DB_GIN".GIN[#si_GIN].FedEx.HLCDataText := #sUDT_RA.HLCDataText;
	            "DB_GIN".GIN[#si_GIN].FedEx.Barcodedata := #sUDT_RA.Barcodedata;
	            "DB_GIN".GIN[#si_GIN].FedEx.HLCResultCode := #sUDT_RA.HLCResultCode;
	        END_IF;
	    END_IF;
	END_REGION

	REGION 6 - Heartbeat Signal
	    // Message is read and type is HB
	    IF #tx_MsgRead
	        AND #sUDT_MSGHeader.MessageType = #cs_HB
	    THEN
	        #iqx_HeartbeatOk := TRUE;

	    END_IF;
	END_REGION
END_FUNCTION_BLOCK

